Universal Robots PolyScope program: 2024DragonThinMarker.urp

Program 2024DragonThinMarker (installation=default directory=/programs createdIn=5.11.9.1010452 lastSavedIn=5.11.9.1010452 robotSerialNumber=20225200364)
Calibrated DH parameters: a=[0.00002, -0.569483, -0.54992, -0.00001, -0.000036, 0]; d=[0.180894, -146.691669, 192.918669, -46.053088, 0.119778, 0.115602]; alpha=[1.571425, -0.001534, 0.003359, 1.568739, -1.571477, 0]; deltaTheta=[0, 0.376258, -0.101074, -0.275185, -0.000002, 0]
Robot Program (runOnlyOnce=true)
  Script file /programs/usbdisk/new-robot/2024Dagonv3_1_thin_marker_large_2.script
    | def Machining1():
    |   # Default parameters:
    |   global speed_ms = 0.3
    |   global speed_rads = 0.75
    |   global accel_mss = 3
    |   global accel_radss = 1.2
    |   global blend_radius_m = 0.001
    | 
    |   # Add subprograms here
    |   # Start of main program
    |   # Program generated by RoboDK v5.6.5 for UR10e on 12/01/2024 13:40:53
    |   # Using nominal kinematics.
    |   blend_radius_m = 0.000
    |   speed_ms = 1.000
    |   # set_reference(p[0.335000, -0.152000, -0.010500, 0.000000, 0.000000, 0.000000])
    |   set_tcp(p[0.000000, 0.000000, 0.252000, 0.000000, 0.000000, 0.000000])
    |   # Show Tool
    |   movej([0.067194, -1.003010, -2.503941, -1.205438, 1.570796, 1.637990],accel_radss,speed_rads,0,blend_radius_m)
    |   movel([0.067194, -1.003010, -2.503941, -1.205438, 1.570796, 1.637990],accel_mss,speed_ms,0,blend_radius_m)
    |   # Splitting Linear movement in 22 (instruction 7: MoveL 3)
    |   movel([0.067194, -1.007550, -2.510737, -1.194102, 1.570796, 1.637990],accel_mss,speed_ms,0,blend_radius_m)
    |   movel([0.067194, -1.012266, -2.517496, -1.182627, 1.570796, 1.637990],accel_mss,speed_ms,0,blend_radius_m)
    |   movel([0.067194, -1.017163, -2.524216, -1.171010, 1.570796, 1.637990],accel_mss,speed_ms,0,blend_radius_m)
    |   movel([0.067194, -1.022245, -2.530898, -1.159246, 1.570796, 1.637990],accel_mss,speed_ms,0,blend_radius_m)
    |   movel([0.067194, -1.027517, -2.537540, -1.147332, 1.570796, 1.637990],accel_mss,speed_ms,0,blend_radius_m)
    |   movel([0.067194, -1.032983, -2.544142, -1.135264, 1.570796, 1.637990],accel_mss,speed_ms,0,blend_radius_m)
    |   movel([0.067194, -1.038648, -2.550703, -1.123038, 1.570796, 1.637990],accel_mss,speed_ms,0,blend_radius_m)
    |   movel([0.067194, -1.044517, -2.557222, -1.110650, 1.570796, 1.637990],accel_mss,speed_ms,0,blend_radius_m)
    |   movel([0.067194, -1.050595, -2.563697, -1.098097, 1.570796, 1.637990],accel_mss,speed_ms,0,blend_radius_m)
    |   movel([0.067194, -1.056888, -2.570128, -1.085374, 1.570796, 1.637990],accel_mss,speed_ms,0,blend_radius_m)
    |   movel([0.067194, -1.063399, -2.576514, -1.072476, 1.570796, 1.637990],accel_mss,speed_ms,0,blend_radius_m)
    |   movel([0.067194, -1.070135, -2.582853, -1.059401, 1.570796, 1.637990],accel_mss,speed_ms,0,blend_radius_m)
    |   movel([0.067194, -1.077101, -2.589145, -1.046144, 1.570796, 1.637990],accel_mss,speed_ms,0,blend_radius_m)
    |   movel([0.067194, -1.084302, -2.595388, -1.032699, 1.570796, 1.637990],accel_mss,speed_ms,0,blend_radius_m)
    |   movel([0.067194, -1.091744, -2.601581, -1.019064, 1.570796, 1.637990],accel_mss,speed_ms,0,blend_radius_m)
    |   movel([0.067194, -1.099433, -2.607722, -1.005234, 1.570796, 1.637990],accel_mss,speed_ms,0,blend_radius_m)
    |   movel([0.067194, -1.107374, -2.613811, -0.991204, 1.570796, 1.637990],accel_mss,speed_ms,0,blend_radius_m)
    |   movel([0.067194, -1.115573, -2.619846, -0.976970, 1.570796, 1.637990],accel_mss,speed_ms,0,blend_radius_m)
    |   movel([0.067194, -1.124036, -2.625825, -0.962528, 1.570796, 1.637990],accel_mss,speed_ms,0,blend_radius_m)
    |   movel([0.067194, -1.132769, -2.631747, -0.947873, 1.570796, 1.637990],accel_mss,speed_ms,0,blend_radius_m)
    |   movel([0.067194, -1.141778, -2.637610, -0.933001, 1.570796, 1.637990],accel_mss,speed_ms,0,blend_radius_m)
    |   movel([0.067194, -1.151068, -2.643412, -0.917908, 1.570796, 1.637990],accel_mss,speed_ms,0,blend_radius_m)
    |   movel([0.067194, -1.151068, -2.643412, -0.917908, 1.570796, 1.637990],accel_mss,speed_ms,0,blend_radius_m)
    |   speed_ms = 1.000
    |   movel([0.067194, -1.151068, -2.643412, -0.917908, 1.570796, 1.637990],accel_mss,speed_ms,0,blend_radius_m)
    |   movel([0.067194, -1.151068, -2.643412, -0.917908, 1.570796, 1.637990],accel_mss,speed_ms,0,blend_radius_m)
    |   movel([0.067194, -1.151068, -2.643412, -0.917908, 1.570796, 1.637990],accel_mss,speed_ms,0,blend_radius_m)
    |   speed_ms = 0.005
    |   # Splitting Linear movement in 4 (instruction 14: MoveL 8)
    |   movel([0.067194, -1.140864, -2.637026, -0.934498, 1.570796, 1.637990],accel_mss,speed_ms,0,blend_radius_m)
    |   movel([0.067194, -1.131001, -2.630567, -0.950821, 1.570796, 1.637990],accel_mss,speed_ms,0,blend_radius_m)
    |   movel([0.067194, -1.121469, -2.624037, -0.966883, 1.570796, 1.637990],accel_mss,speed_ms,0,blend_radius_m)
    |   movel([0.067194, -1.112262, -2.617439, -0.982688, 1.570796, 1.637990],accel_mss,speed_ms,0,blend_radius_m)
    |   speed_ms = 1.000
    |   # Splitting Linear movement in 4 (instruction 16: MoveL 9)
    |   movel([0.067194, -1.121469, -2.624037, -0.966883, 1.570796, 1.637990],accel_mss,speed_ms,0,blend_radius_m)
    |   movel([0.067194, -1.131001, -2.630567, -0.950821, 1.570796, 1.637990],accel_mss,speed_ms,0,blend_radius_m)
    |   movel([0.067194, -1.140864, -2.637026, -0.934498, 1.570796, 1.637990],accel_mss,speed_ms,0,blend_radius_m)
    |   movel([0.067194, -1.151068, -2.643412, -0.917908, 1.570796, 1.637990],accel_mss,speed_ms,0,blend_radius_m)
    |   speed_ms = 0.040
    |   movel([0.067194, -1.151068, -2.643412, -0.917908, 1.570796, 1.637990],accel_mss,speed_ms,0,blend_radius_m)
    |   speed_ms = 1.000
    |   movel([0.067194, -1.151068, -2.643412, -0.917908, 1.570796, 1.637990],accel_mss,speed_ms,0,blend_radius_m)
    |   # Splitting Linear movement in 16 (instruction 21: MoveL 12)
    |   movel([0.074500, -1.158538, -2.640023, -0.913828, 1.570796, 1.645297],accel_mss,speed_ms,0,blend_radius_m)
    |   movel([0.081655, -1.166054, -2.636556, -0.909779, 1.570796, 1.652452],accel_mss,speed_ms,0,blend_radius_m)
    |   movel([0.088662, -1.173611, -2.633012, -0.905766, 1.570796, 1.659459],accel_mss,speed_ms,0,blend_radius_m)
    |   movel([0.095525, -1.181205, -2.629391, -0.901793, 1.570796, 1.666321],accel_mss,speed_ms,0,blend_radius_m)
    |   movel([0.102245, -1.188830, -2.625693, -0.897865, 1.570796, 1.673041],accel_mss,speed_ms,0,blend_radius_m)
    |   movel([0.108826, -1.196483, -2.621921, -0.893985, 1.570796, 1.679622],accel_mss,speed_ms,0,blend_radius_m)
    |   movel([0.115271, -1.204158, -2.618073, -0.890157, 1.570796, 1.686068],accel_mss,speed_ms,0,blend_radius_m)
    |   movel([0.121584, -1.211853, -2.614152, -0.886384, 1.570796, 1.692381],accel_mss,speed_ms,0,blend_radius_m)
    |   movel([0.127767, -1.219562, -2.610158, -0.882669, 1.570796, 1.698563],accel_mss,speed_ms,0,blend_radius_m)
    |   movel([0.133823, -1.227283, -2.606091, -0.879015, 1.570796, 1.704619],accel_mss,speed_ms,0,blend_radius_m)
    |   movel([0.139755, -1.235012, -2.601952, -0.875425, 1.570796, 1.710551],accel_mss,speed_ms,0,blend_radius_m)
    |   movel([0.145566, -1.242745, -2.597743, -0.871901, 1.570796, 1.716362],accel_mss,speed_ms,0,blend_radius_m)
    |   movel([0.151258, -1.250480, -2.593464, -0.868445, 1.570796, 1.722054],accel_mss,speed_ms,0,blend_radius_m)
    |   movel([0.156835, -1.258213, -2.589116, -0.865060, 1.570796, 1.727631],accel_mss,speed_ms,0,blend_radius_m)
    |   movel([0.162299, -1.265943, -2.584700, -0.861746, 1.570796, 1.733095],accel_mss,speed_ms,0,blend_radius_m)
    |   movel([0.167652, -1.273666, -2.580216, -0.858507, 1.570796, 1.738448],accel_mss,speed_ms,0,blend_radius_m)
    |   speed_ms = 0.005
    |   # Splitting Linear movement in 4 (instruction 23: MoveL 13)
    |   movel([0.167652, -1.283824, -2.585872, -0.842693, 1.570796, 1.738448],accel_mss,speed_ms,0,blend_radius_m)
    |   movel([0.167652, -1.294258, -2.591445, -0.826686, 1.570796, 1.738448],accel_mss,speed_ms,0,blend_radius_m)
    |   movel([0.167652, -1.304973, -2.596930, -0.810486, 1.570796, 1.738448],accel_mss,speed_ms,0,blend_radius_m)
    |   movel([0.167652, -1.315971, -2.602326, -0.794092, 1.570796, 1.738448],accel_mss,speed_ms,0,blend_radius_m)
    |   speed_ms = 0.035
    |   movel([0.173157, -1.309286, -2.606449, -0.796654, 1.570796, 1.743953],accel_mss,speed_ms,0,blend_radius_m)
    |   movel([0.180818, -1.304394, -2.609429, -0.798566, 1.570796, 1.751614],accel_mss,speed_ms,0,blend_radius_m)
    |   movel([0.187193, -1.302810, -2.610387, -0.799192, 1.570796, 1.757989],accel_mss,speed_ms,0,blend_radius_m)
    |   movel([0.192434, -1.303607, -2.609905, -0.798877, 1.570796, 1.763230],accel_mss,speed_ms,0,blend_radius_m)
    |   movel([0.197299, -1.311355, -2.605179, -0.795855, 1.570796, 1.768095],accel_mss,speed_ms,0,blend_radius_m)
    |   movel([0.196080, -1.317152, -2.601592, -0.793645, 1.570796, 1.766876],accel_mss,speed_ms,0,blend_radius_m)
    |   movel([0.187692, -1.327691, -2.594957, -0.789741, 1.570796, 1.758489],accel_mss,speed_ms,0,blend_radius_m)
    |   movel([0.181558, -1.331218, -2.592703, -0.788467, 1.570796, 1.752354],accel_mss,speed_ms,0,blend_radius_m)
    |   movel([0.173175, -1.332644, -2.591788, -0.787957, 1.570796, 1.743971],accel_mss,speed_ms,0,blend_radius_m)
    |   speed_ms = 0.005
    |   movel([0.173175, -1.323918, -2.587552, -0.800919, 1.570796, 1.743971],accel_mss,speed_ms,0,blend_radius_m)
    |   speed_ms = 0.040
    |   # Splitting Linear movement in 4 (instruction 37: MoveL 24)
    |   movel([0.168800, -1.330792, -2.583155, -0.798442, 1.570796, 1.739596],accel_mss,speed_ms,0,blend_radius_m)
    |   movel([0.164486, -1.337594, -2.578742, -0.796052, 1.570796, 1.735282],accel_mss,speed_ms,0,blend_radius_m)
    |   movel([0.160232, -1.344326, -2.574314, -0.793749, 1.570796, 1.731029],accel_mss,speed_ms,0,blend_radius_m)
    |   movel([0.156038, -1.350989, -2.569871, -0.791529, 1.570796, 1.726834],accel_mss,speed_ms,0,blend_radius_m)
    |   speed_ms = 0.005
    |   movel([0.156038, -1.359551, -2.573989, -0.778848, 1.570796, 1.726834],accel_mss,speed_ms,0,blend_radius_m)
    |   speed_ms = 0.035
    |   movel([0.156883, -1.369330, -2.567274, -0.775785, 1.570796, 1.727679],accel_mss,speed_ms,0,blend_radius_m)
    |   movel([0.154042, -1.379446, -2.560185, -0.772758, 1.570796, 1.724839],accel_mss,speed_ms,0,blend_radius_m)
    |   movel([0.147953, -1.388965, -2.553382, -0.770042, 1.570796, 1.718749],accel_mss,speed_ms,0,blend_radius_m)
    |   movel([0.138991, -1.397044, -2.547506, -0.767839, 1.570796, 1.709787],accel_mss,speed_ms,0,blend_radius_m)
    |   movel([0.127521, -1.402604, -2.543408, -0.766378, 1.570796, 1.698317],accel_mss,speed_ms,0,blend_radius_m)
    |   movel([0.118961, -1.405060, -2.541583, -0.765746, 1.570796, 1.689757],accel_mss,speed_ms,0,blend_radius_m)
    |   speed_ms = 0.005
    |   movel([0.118961, -1.396797, -2.537660, -0.777932, 1.570796, 1.689757],accel_mss,speed_ms,0,blend_radius_m)
    |   speed_ms = 0.040
    |   # Splitting Linear movement in 2 (instruction 50: MoveL 33)
    |   movel([0.112287, -1.401146, -2.534448, -0.776795, 1.570796, 1.683083],accel_mss,speed_ms,0,blend_radius_m)
    |   movel([0.105663, -1.405490, -2.531212, -0.775687, 1.570796, 1.676460],accel_mss,speed_ms,0,blend_radius_m)
    |   speed_ms = 0.005
    |   movel([0.105663, -1.413694, -2.535098, -0.763597, 1.570796, 1.676460],accel_mss,speed_ms,0,blend_radius_m)
    |   speed_ms = 0.035
    |   movel([0.101650, -1.423004, -2.527983, -0.761402, 1.570796, 1.672447],accel_mss,speed_ms,0,blend_radius_m)
    |   movel([0.104946, -1.429410, -2.523012, -0.759967, 1.570796, 1.675742],accel_mss,speed_ms,0,blend_radius_m)
    |   movel([0.113388, -1.430242, -2.522362, -0.759785, 1.570796, 1.684184],accel_mss,speed_ms,0,blend_radius_m)
    |   movel([0.118946, -1.427701, -2.524344, -0.760344, 1.570796, 1.689742],accel_mss,speed_ms,0,blend_radius_m)
    |   movel([0.125116, -1.422682, -2.528231, -0.761476, 1.570796, 1.695912],accel_mss,speed_ms,0,blend_radius_m)
    |   speed_ms = 0.005
    |   movel([0.125116, -1.414541, -2.524382, -0.773466, 1.570796, 1.695912],accel_mss,speed_ms,0,blend_radius_m)
    |   speed_ms = 0.040
    |   # Splitting Linear movement in 6 (instruction 62: MoveL 41)
    |   movel([0.131385, -1.420188, -2.520061, -0.772140, 1.570796, 1.702182],accel_mss,speed_ms,0,blend_radius_m)
    |   movel([0.137555, -1.425859, -2.515674, -0.770856, 1.570796, 1.708351],accel_mss,speed_ms,0,blend_radius_m)
    |   movel([0.143625, -1.431553, -2.511222, -0.769614, 1.570796, 1.714422],accel_mss,speed_ms,0,blend_radius_m)
    |   movel([0.149599, -1.437267, -2.506705, -0.768417, 1.570796, 1.720395],accel_mss,speed_ms,0,blend_radius_m)
    |   movel([0.155477, -1.443000, -2.502125, -0.767263, 1.570796, 1.726274],accel_mss,speed_ms,0,blend_radius_m)
    |   movel([0.161262, -1.448750, -2.497482, -0.766156, 1.570796, 1.732058],accel_mss,speed_ms,0,blend_radius_m)
    |   speed_ms = 0.005
    |   movel([0.161262, -1.456649, -2.501190, -0.754550, 1.570796, 1.732058],accel_mss,speed_ms,0,blend_radius_m)
    |   speed_ms = 0.035
    |   # Splitting Linear movement in 4 (instruction 66: MoveL 43)
    |   movel([0.152429, -1.458352, -2.499789, -0.754248, 1.570796, 1.723226],accel_mss,speed_ms,0,blend_radius_m)
    |   movel([0.143603, -1.460114, -2.498334, -0.753941, 1.570796, 1.714400],accel_mss,speed_ms,0,blend_radius_m)
    |   movel([0.134785, -1.461934, -2.496827, -0.753628, 1.570796, 1.705581],accel_mss,speed_ms,0,blend_radius_m)
    |   movel([0.125976, -1.463810, -2.495267, -0.753312, 1.570796, 1.696772],accel_mss,speed_ms,0,blend_radius_m)
    |   # Splitting Linear movement in 4 (instruction 67: MoveL 44)
    |   movel([0.130374, -1.457124, -2.500800, -0.754465, 1.570796, 1.701171],accel_mss,speed_ms,0,blend_radius_m)
    |   movel([0.134837, -1.450374, -2.506316, -0.755698, 1.570796, 1.705633],accel_mss,speed_ms,0,blend_radius_m)
    |   movel([0.139366, -1.443560, -2.511816, -0.757013, 1.570796, 1.710162],accel_mss,speed_ms,0,blend_radius_m)
    |   movel([0.143961, -1.436680, -2.517298, -0.758412, 1.570796, 1.714758],accel_mss,speed_ms,0,blend_radius_m)
    |   movel([0.147089, -1.433429, -2.519863, -0.759097, 1.570796, 1.717886],accel_mss,speed_ms,0,blend_radius_m)
    |   movel([0.150947, -1.432131, -2.520882, -0.759376, 1.570796, 1.721743],accel_mss,speed_ms,0,blend_radius_m)
    |   movel([0.155136, -1.432926, -2.520258, -0.759205, 1.570796, 1.725933],accel_mss,speed_ms,0,blend_radius_m)
    |   movel([0.156013, -1.436691, -2.517289, -0.758410, 1.570796, 1.726809],accel_mss,speed_ms,0,blend_radius_m)
    |   # Splitting Linear movement in 2 (instruction 72: MoveL 49)
    |   movel([0.154617, -1.445524, -2.510238, -0.756627, 1.570796, 1.725413],accel_mss,speed_ms,0,blend_radius_m)
    |   movel([0.153250, -1.454249, -2.503159, -0.754982, 1.570796, 1.724046],accel_mss,speed_ms,0,blend_radius_m)
    |   speed_ms = 0.005
    |   movel([0.153250, -1.446333, -2.499441, -0.766616, 1.570796, 1.724046],accel_mss,speed_ms,0,blend_radius_m)
    |   speed_ms = 0.040
    |   # Splitting Linear movement in 4 (instruction 76: MoveL 51)
    |   movel([0.146625, -1.442667, -2.502393, -0.767329, 1.570796, 1.717422],accel_mss,speed_ms,0,blend_radius_m)
    |   movel([0.139925, -1.439047, -2.505289, -0.768053, 1.570796, 1.710722],accel_mss,speed_ms,0,blend_radius_m)
    |   movel([0.133149, -1.435473, -2.508129, -0.768787, 1.570796, 1.703945],accel_mss,speed_ms,0,blend_radius_m)
    |   movel([0.126295, -1.431947, -2.510912, -0.769530, 1.570796, 1.697092],accel_mss,speed_ms,0,blend_radius_m)
    |   speed_ms = 0.005
    |   movel([0.126295, -1.439966, -2.514688, -0.757735, 1.570796, 1.697092],accel_mss,speed_ms,0,blend_radius_m)
    |   speed_ms = 0.035
    |   # Splitting Linear movement in 4 (instruction 80: MoveL 53)
    |   movel([0.120303, -1.448950, -2.507472, -0.755967, 1.570796, 1.691099],accel_mss,speed_ms,0,blend_radius_m)
    |   movel([0.114424, -1.457822, -2.500226, -0.754341, 1.570796, 1.685220],accel_mss,speed_ms,0,blend_radius_m)
    |   movel([0.108656, -1.466585, -2.492951, -0.752853, 1.570796, 1.679453],accel_mss,speed_ms,0,blend_radius_m)
    |   movel([0.102997, -1.475244, -2.485647, -0.751498, 1.570796, 1.673793],accel_mss,speed_ms,0,blend_radius_m)
    |   speed_ms = 0.005
    |   movel([0.102997, -1.467481, -2.482014, -0.762894, 1.570796, 1.673793],accel_mss,speed_ms,0,blend_radius_m)
    |   speed_ms = 0.040
    |   movel([0.108909, -1.471851, -2.478329, -0.762209, 1.570796, 1.679706],accel_mss,speed_ms,0,blend_radius_m)
    |   speed_ms = 0.005
    |   movel([0.108909, -1.479582, -2.481945, -0.750863, 1.570796, 1.679706],accel_mss,speed_ms,0,blend_radius_m)
    |   speed_ms = 0.035
    |   # Splitting Linear movement in 6 (instruction 88: MoveL 57)
    |   movel([0.117333, -1.477702, -2.483553, -0.751135, 1.570796, 1.688130],accel_mss,speed_ms,0,blend_radius_m)
    |   movel([0.125768, -1.475873, -2.485112, -0.751404, 1.570796, 1.696564],accel_mss,speed_ms,0,blend_radius_m)
    |   movel([0.134212, -1.474095, -2.486622, -0.751671, 1.570796, 1.705008],accel_mss,speed_ms,0,blend_radius_m)
    |   movel([0.142664, -1.472370, -2.488083, -0.751935, 1.570796, 1.713461],accel_mss,speed_ms,0,blend_radius_m)
    |   movel([0.151124, -1.470699, -2.489495, -0.752195, 1.570796, 1.721920],accel_mss,speed_ms,0,blend_radius_m)
    |   movel([0.159589, -1.469080, -2.490858, -0.752451, 1.570796, 1.730386],accel_mss,speed_ms,0,blend_radius_m)
    |   speed_ms = 0.005
    |   movel([0.159589, -1.461273, -2.487200, -0.763916, 1.570796, 1.730386],accel_mss,speed_ms,0,blend_radius_m)
    |   speed_ms = 0.040
    |   movel([0.149536, -1.467349, -2.482125, -0.762915, 1.570796, 1.720332],accel_mss,speed_ms,0,blend_radius_m)
    |   speed_ms = 0.005
    |   movel([0.149536, -1.475113, -2.485758, -0.751518, 1.570796, 1.720332],accel_mss,speed_ms,0,blend_radius_m)
    |   speed_ms = 0.035
    |   # Splitting Linear movement in 2 (instruction 96: MoveL 61)
    |   movel([0.148238, -1.482664, -2.479296, -0.750429, 1.570796, 1.719034],accel_mss,speed_ms,0,blend_radius_m)
    |   movel([0.146962, -1.490139, -2.472812, -0.749438, 1.570796, 1.717758],accel_mss,speed_ms,0,blend_radius_m)
    |   speed_ms = 0.005
    |   movel([0.146962, -1.482487, -2.469238, -0.760664, 1.570796, 1.717758],accel_mss,speed_ms,0,blend_radius_m)
    |   speed_ms = 0.040
    |   # Splitting Linear movement in 4 (instruction 100: MoveL 63)
    |   movel([0.148044, -1.489667, -2.463003, -0.759718, 1.570796, 1.718840],accel_mss,speed_ms,0,blend_radius_m)
    |   movel([0.149106, -1.496792, -2.456739, -0.758858, 1.570796, 1.719903],accel_mss,speed_ms,0,blend_radius_m)
    |   movel([0.150151, -1.503862, -2.450444, -0.758082, 1.570796, 1.720947],accel_mss,speed_ms,0,blend_radius_m)
    |   movel([0.151177, -1.510880, -2.444121, -0.757388, 1.570796, 1.721973],accel_mss,speed_ms,0,blend_radius_m)
    |   speed_ms = 0.005
    |   movel([0.151177, -1.518320, -2.447586, -0.746483, 1.570796, 1.721973],accel_mss,speed_ms,0,blend_radius_m)
    |   speed_ms = 0.035
    |   movel([0.144185, -1.518298, -2.447607, -0.746484, 1.570796, 1.714981],accel_mss,speed_ms,0,blend_radius_m)
    |   movel([0.135810, -1.523039, -2.443241, -0.746109, 1.570796, 1.706606],accel_mss,speed_ms,0,blend_radius_m)
    |   speed_ms = 0.005
    |   movel([0.135810, -1.515634, -2.439793, -0.756962, 1.570796, 1.706606],accel_mss,speed_ms,0,blend_radius_m)
    |   speed_ms = 0.040
    |   # Splitting Linear movement in 2 (instruction 109: MoveL 68)
    |   movel([0.131950, -1.512601, -2.442559, -0.757230, 1.570796, 1.702747],accel_mss,speed_ms,0,blend_radius_m)
    |   movel([0.128057, -1.509579, -2.445299, -0.757511, 1.570796, 1.698854],accel_mss,speed_ms,0,blend_radius_m)
    |   speed_ms = 0.005
    |   movel([0.128057, -1.517029, -2.448769, -0.746591, 1.570796, 1.698854],accel_mss,speed_ms,0,blend_radius_m)
    |   speed_ms = 0.035
    |   movel([0.135688, -1.510985, -2.454272, -0.747132, 1.570796, 1.706484],accel_mss,speed_ms,0,blend_radius_m)
    |   movel([0.145709, -1.507599, -2.457330, -0.747461, 1.570796, 1.716505],accel_mss,speed_ms,0,blend_radius_m)
    |   movel([0.153057, -1.507247, -2.457646, -0.747496, 1.570796, 1.723854],accel_mss,speed_ms,0,blend_radius_m)
    |   movel([0.160779, -1.504715, -2.459919, -0.747754, 1.570796, 1.731575],accel_mss,speed_ms,0,blend_radius_m)
    |   movel([0.165697, -1.498711, -2.465270, -0.748408, 1.570796, 1.736494],accel_mss,speed_ms,0,blend_radius_m)
    |   movel([0.165769, -1.494615, -2.468888, -0.748886, 1.570796, 1.736565],accel_mss,speed_ms,0,blend_radius_m)
    |   movel([0.161795, -1.491118, -2.471957, -0.749314, 1.570796, 1.732592],accel_mss,speed_ms,0,blend_radius_m)
    |   speed_ms = 0.005
    |   movel([0.161795, -1.483474, -2.468386, -0.760529, 1.570796, 1.732592],accel_mss,speed_ms,0,blend_radius_m)
    |   speed_ms = 0.040
    |   movel([0.163598, -1.478856, -2.472361, -0.761172, 1.570796, 1.734394],accel_mss,speed_ms,0,blend_radius_m)
    |   speed_ms = 0.005
    |   movel([0.163598, -1.486535, -2.475950, -0.749905, 1.570796, 1.734394],accel_mss,speed_ms,0,blend_radius_m)
    |   speed_ms = 0.035
    |   # Splitting Linear movement in 6 (instruction 127: MoveL 80)
    |   movel([0.165237, -1.477873, -2.483407, -0.751110, 1.570796, 1.736033],accel_mss,speed_ms,0,blend_radius_m)
    |   movel([0.166909, -1.469106, -2.490836, -0.752447, 1.570796, 1.737705],accel_mss,speed_ms,0,blend_radius_m)
    |   movel([0.168617, -1.460232, -2.498236, -0.753920, 1.570796, 1.739413],accel_mss,speed_ms,0,blend_radius_m)
    |   movel([0.170360, -1.451246, -2.505608, -0.755535, 1.570796, 1.741157],accel_mss,speed_ms,0,blend_radius_m)
    |   movel([0.172141, -1.442144, -2.512950, -0.757295, 1.570796, 1.742938],accel_mss,speed_ms,0,blend_radius_m)
    |   movel([0.173961, -1.432921, -2.520262, -0.759206, 1.570796, 1.744757],accel_mss,speed_ms,0,blend_radius_m)
    |   movel([0.174121, -1.425301, -2.526207, -0.760881, 1.570796, 1.744918],accel_mss,speed_ms,0,blend_radius_m)
    |   movel([0.171855, -1.420034, -2.530266, -0.762089, 1.570796, 1.742651],accel_mss,speed_ms,0,blend_radius_m)
    |   movel([0.164710, -1.415086, -2.534042, -0.763261, 1.570796, 1.735506],accel_mss,speed_ms,0,blend_radius_m)
    |   movel([0.157581, -1.414562, -2.534440, -0.763387, 1.570796, 1.728377],accel_mss,speed_ms,0,blend_radius_m)
    |   movel([0.149868, -1.416547, -2.532931, -0.762911, 1.570796, 1.720665],accel_mss,speed_ms,0,blend_radius_m)
    |   # Splitting Linear movement in 2 (instruction 133: MoveL 86)
    |   movel([0.143461, -1.420629, -2.529810, -0.761950, 1.570796, 1.714257],accel_mss,speed_ms,0,blend_radius_m)
    |   movel([0.137100, -1.424708, -2.526667, -0.761015, 1.570796, 1.707896],accel_mss,speed_ms,0,blend_radius_m)
    |   # Splitting Linear movement in 2 (instruction 134: MoveL 87)
    |   movel([0.131353, -1.430632, -2.522057, -0.759700, 1.570796, 1.702149],accel_mss,speed_ms,0,blend_radius_m)
    |   movel([0.125674, -1.436514, -2.517428, -0.758446, 1.570796, 1.696470],accel_mss,speed_ms,0,blend_radius_m)
    |   movel([0.119296, -1.440811, -2.514015, -0.757564, 1.570796, 1.690092],accel_mss,speed_ms,0,blend_radius_m)
    |   movel([0.110431, -1.444256, -2.511257, -0.756876, 1.570796, 1.681228],accel_mss,speed_ms,0,blend_radius_m)
    |   movel([0.101817, -1.445410, -2.510330, -0.756649, 1.570796, 1.672613],accel_mss,speed_ms,0,blend_radius_m)
    |   movel([0.094928, -1.444091, -2.511390, -0.756908, 1.570796, 1.665724],accel_mss,speed_ms,0,blend_radius_m)
    |   # Splitting Linear movement in 2 (instruction 139: MoveL 92)
    |   movel([0.090922, -1.441165, -2.513732, -0.757492, 1.570796, 1.661719],accel_mss,speed_ms,0,blend_radius_m)
    |   movel([0.086882, -1.438253, -2.516050, -0.758086, 1.570796, 1.657679],accel_mss,speed_ms,0,blend_radius_m)
    |   # Splitting Linear movement in 2 (instruction 140: MoveL 93)
    |   movel([0.085417, -1.432512, -2.520583, -0.759294, 1.570796, 1.656214],accel_mss,speed_ms,0,blend_radius_m)
    |   movel([0.083931, -1.426737, -2.525094, -0.760558, 1.570796, 1.654728],accel_mss,speed_ms,0,blend_radius_m)
    |   # Splitting Linear movement in 2 (instruction 141: MoveL 94)
    |   movel([0.085999, -1.420689, -2.529764, -0.761936, 1.570796, 1.656796],accel_mss,speed_ms,0,blend_radius_m)
    |   movel([0.088096, -1.414585, -2.534422, -0.763381, 1.570796, 1.658892],accel_mss,speed_ms,0,blend_radius_m)
    |   # Splitting Linear movement in 2 (instruction 142: MoveL 95)
    |   movel([0.092936, -1.409123, -2.538545, -0.764721, 1.570796, 1.663732],accel_mss,speed_ms,0,blend_radius_m)
    |   movel([0.097830, -1.403621, -2.542653, -0.766115, 1.570796, 1.668626],accel_mss,speed_ms,0,blend_radius_m)
    |   # Splitting Linear movement in 2 (instruction 143: MoveL 96)
    |   movel([0.104573, -1.399755, -2.545513, -0.767121, 1.570796, 1.675370],accel_mss,speed_ms,0,blend_radius_m)
    |   movel([0.111360, -1.395891, -2.548350, -0.768147, 1.570796, 1.682157],accel_mss,speed_ms,0,blend_radius_m)
    |   speed_ms = 0.005
    |   movel([0.111360, -1.387566, -2.544389, -0.780434, 1.570796, 1.682157],accel_mss,speed_ms,0,blend_radius_m)
    |   speed_ms = 0.040
    |   movel([0.119864, -1.383368, -2.547408, -0.781612, 1.570796, 1.690661],accel_mss,speed_ms,0,blend_radius_m)
    |   speed_ms = 0.005
    |   movel([0.119864, -1.391722, -2.551388, -0.769280, 1.570796, 1.690661],accel_mss,speed_ms,0,blend_radius_m)
    |   speed_ms = 0.035
    |   movel([0.127885, -1.389591, -2.552930, -0.769868, 1.570796, 1.698681],accel_mss,speed_ms,0,blend_radius_m)
    |   movel([0.133367, -1.385898, -2.555588, -0.770903, 1.570796, 1.704163],accel_mss,speed_ms,0,blend_radius_m)
    |   movel([0.139947, -1.375961, -2.562643, -0.773785, 1.570796, 1.710744],accel_mss,speed_ms,0,blend_radius_m)
    |   movel([0.140218, -1.370886, -2.566192, -0.775310, 1.570796, 1.711014],accel_mss,speed_ms,0,blend_radius_m)
    |   movel([0.134172, -1.364852, -2.570365, -0.777171, 1.570796, 1.704969],accel_mss,speed_ms,0,blend_radius_m)
    |   movel([0.128886, -1.364770, -2.570422, -0.777197, 1.570796, 1.699682],accel_mss,speed_ms,0,blend_radius_m)
    |   movel([0.122870, -1.366828, -2.569005, -0.776556, 1.570796, 1.693666],accel_mss,speed_ms,0,blend_radius_m)
    |   movel([0.116129, -1.371828, -2.565537, -0.775024, 1.570796, 1.686926],accel_mss,speed_ms,0,blend_radius_m)
    |   movel([0.111791, -1.378110, -2.561130, -0.773150, 1.570796, 1.682587],accel_mss,speed_ms,0,blend_radius_m)
    |   speed_ms = 0.005
    |   movel([0.111791, -1.369666, -2.557092, -0.785631, 1.570796, 1.682587],accel_mss,speed_ms,0,blend_radius_m)
    |   speed_ms = 0.040
    |   # Splitting Linear movement in 2 (instruction 163: MoveL 110)
    |   movel([0.102143, -1.369221, -2.557402, -0.785766, 1.570796, 1.672940],accel_mss,speed_ms,0,blend_radius_m)
    |   movel([0.092446, -1.368873, -2.557645, -0.785872, 1.570796, 1.663242],accel_mss,speed_ms,0,blend_radius_m)
    |   speed_ms = 0.005
    |   movel([0.092446, -1.377321, -2.561686, -0.773382, 1.570796, 1.663242],accel_mss,speed_ms,0,blend_radius_m)
    |   speed_ms = 0.035
    |   # Splitting Linear movement in 2 (instruction 167: MoveL 112)
    |   movel([0.096801, -1.371069, -2.566066, -0.775255, 1.570796, 1.667598],accel_mss,speed_ms,0,blend_radius_m)
    |   movel([0.101214, -1.364757, -2.570431, -0.777201, 1.570796, 1.672011],accel_mss,speed_ms,0,blend_radius_m)
    |   movel([0.109892, -1.356186, -2.576270, -0.779933, 1.570796, 1.680688],accel_mss,speed_ms,0,blend_radius_m)
    |   # Splitting Linear movement in 2 (instruction 169: MoveL 114)
    |   movel([0.116564, -1.352214, -2.578941, -0.781234, 1.570796, 1.687360],accel_mss,speed_ms,0,blend_radius_m)
    |   movel([0.123279, -1.348242, -2.581591, -0.782556, 1.570796, 1.694075],accel_mss,speed_ms,0,blend_radius_m)
    |   # Splitting Linear movement in 2 (instruction 170: MoveL 115)
    |   movel([0.130460, -1.346443, -2.582783, -0.783162, 1.570796, 1.701256],accel_mss,speed_ms,0,blend_radius_m)
    |   movel([0.137648, -1.344681, -2.583948, -0.783760, 1.570796, 1.708444],accel_mss,speed_ms,0,blend_radius_m)
    |   # Splitting Linear movement in 2 (instruction 171: MoveL 116)
    |   movel([0.147112, -1.346959, -2.582442, -0.782988, 1.570796, 1.717908],accel_mss,speed_ms,0,blend_radius_m)
    |   movel([0.156484, -1.349338, -2.580862, -0.782189, 1.570796, 1.727280],accel_mss,speed_ms,0,blend_radius_m)
    |   movel([0.165265, -1.351727, -2.579267, -0.781395, 1.570796, 1.736061],accel_mss,speed_ms,0,blend_radius_m)
    |   movel([0.175465, -1.350957, -2.579782, -0.781650, 1.570796, 1.746261],accel_mss,speed_ms,0,blend_radius_m)
    |   movel([0.186285, -1.347233, -2.582261, -0.782896, 1.570796, 1.757082],accel_mss,speed_ms,0,blend_radius_m)
    |   movel([0.196943, -1.340710, -2.586556, -0.785123, 1.570796, 1.767739],accel_mss,speed_ms,0,blend_radius_m)
    |   movel([0.205914, -1.332349, -2.591977, -0.788062, 1.570796, 1.776710],accel_mss,speed_ms,0,blend_radius_m)
    |   movel([0.213309, -1.322133, -2.598475, -0.791782, 1.570796, 1.784105],accel_mss,speed_ms,0,blend_radius_m)
    |   movel([0.218019, -1.310769, -2.605539, -0.796081, 1.570796, 1.788815],accel_mss,speed_ms,0,blend_radius_m)
    |   movel([0.218847, -1.299039, -2.612655, -0.800695, 1.570796, 1.789643],accel_mss,speed_ms,0,blend_radius_m)
    |   movel([0.215629, -1.290767, -2.617567, -0.804055, 1.570796, 1.786426],accel_mss,speed_ms,0,blend_radius_m)
    |   movel([0.208938, -1.285368, -2.620726, -0.806295, 1.570796, 1.779735],accel_mss,speed_ms,0,blend_radius_m)
    |   movel([0.199486, -1.283243, -2.621959, -0.807187, 1.570796, 1.770282],accel_mss,speed_ms,0,blend_radius_m)
    |   movel([0.188071, -1.284713, -2.621106, -0.806569, 1.570796, 1.758867],accel_mss,speed_ms,0,blend_radius_m)
    |   movel([0.175553, -1.290033, -2.617999, -0.804358, 1.570796, 1.746349],accel_mss,speed_ms,0,blend_radius_m)
    |   movel([0.164105, -1.298333, -2.613078, -0.800978, 1.570796, 1.734901],accel_mss,speed_ms,0,blend_radius_m)
    |   movel([0.154717, -1.308660, -2.606832, -0.796897, 1.570796, 1.725514],accel_mss,speed_ms,0,blend_radius_m)
    |   movel([0.148273, -1.320113, -2.599743, -0.792533, 1.570796, 1.719069],accel_mss,speed_ms,0,blend_radius_m)
    |   speed_ms = 0.005
    |   movel([0.148273, -1.311314, -2.595451, -0.805623, 1.570796, 1.719069],accel_mss,speed_ms,0,blend_radius_m)
    |   speed_ms = 0.040
    |   movel([0.148587, -1.300615, -2.601996, -0.809778, 1.570796, 1.719384],accel_mss,speed_ms,0,blend_radius_m)
    |   speed_ms = 0.005
    |   movel([0.148587, -1.309472, -2.606335, -0.796582, 1.570796, 1.719384],accel_mss,speed_ms,0,blend_radius_m)
    |   speed_ms = 0.035
    |   # Splitting Linear movement in 2 (instruction 195: MoveL 136)
    |   movel([0.141454, -1.310148, -2.605920, -0.796320, 1.570796, 1.712250],accel_mss,speed_ms,0,blend_radius_m)
    |   movel([0.134308, -1.310872, -2.605476, -0.796041, 1.570796, 1.705104],accel_mss,speed_ms,0,blend_radius_m)
    |   # Splitting Linear movement in 2 (instruction 196: MoveL 137)
    |   movel([0.128832, -1.308947, -2.606656, -0.796786, 1.570796, 1.699629],accel_mss,speed_ms,0,blend_radius_m)
    |   movel([0.123318, -1.307057, -2.607810, -0.797521, 1.570796, 1.694114],accel_mss,speed_ms,0,blend_radius_m)
    |   # Splitting Linear movement in 2 (instruction 197: MoveL 138)
    |   movel([0.119974, -1.302841, -2.610368, -0.799180, 1.570796, 1.690770],accel_mss,speed_ms,0,blend_radius_m)
    |   movel([0.116592, -1.298625, -2.612903, -0.800861, 1.570796, 1.687388],accel_mss,speed_ms,0,blend_radius_m)
    |   # Splitting Linear movement in 2 (instruction 198: MoveL 139)
    |   movel([0.115954, -1.292359, -2.616628, -0.803402, 1.570796, 1.686750],accel_mss,speed_ms,0,blend_radius_m)
    |   movel([0.115306, -1.286042, -2.620333, -0.806014, 1.570796, 1.686102],accel_mss,speed_ms,0,blend_radius_m)
    |   # Splitting Linear movement in 2 (instruction 199: MoveL 140)
    |   movel([0.117736, -1.278694, -2.624580, -0.809115, 1.570796, 1.688532],accel_mss,speed_ms,0,blend_radius_m)
    |   movel([0.120205, -1.271258, -2.628809, -0.812322, 1.570796, 1.691002],accel_mss,speed_ms,0,blend_radius_m)
    |   # Splitting Linear movement in 2 (instruction 200: MoveL 141)
    |   movel([0.125251, -1.264165, -2.632779, -0.815444, 1.570796, 1.696048],accel_mss,speed_ms,0,blend_radius_m)
    |   movel([0.130370, -1.256992, -2.636733, -0.818665, 1.570796, 1.701166],accel_mss,speed_ms,0,blend_radius_m)
    |   # Splitting Linear movement in 2 (instruction 201: MoveL 142)
    |   movel([0.137370, -1.251001, -2.639986, -0.821401, 1.570796, 1.708167],accel_mss,speed_ms,0,blend_radius_m)
    |   movel([0.144445, -1.244971, -2.643219, -0.824200, 1.570796, 1.715241],accel_mss,speed_ms,0,blend_radius_m)
    |   # Splitting Linear movement in 2 (instruction 202: MoveL 143)
    |   movel([0.152629, -1.241031, -2.645307, -0.826051, 1.570796, 1.723426],accel_mss,speed_ms,0,blend_radius_m)
    |   movel([0.160854, -1.237110, -2.647367, -0.827911, 1.570796, 1.731651],accel_mss,speed_ms,0,blend_radius_m)
    |   # Splitting Linear movement in 2 (instruction 203: MoveL 144)
    |   movel([0.170134, -1.236501, -2.647686, -0.828202, 1.570796, 1.740930],accel_mss,speed_ms,0,blend_radius_m)
    |   movel([0.179381, -1.235980, -2.647958, -0.828451, 1.570796, 1.750178],accel_mss,speed_ms,0,blend_radius_m)
    |   speed_ms = 0.005
    |   movel([0.179381, -1.226775, -2.643291, -0.842324, 1.570796, 1.750178],accel_mss,speed_ms,0,blend_radius_m)
    |   speed_ms = 0.040
    |   # Splitting Linear movement in 4 (instruction 207: MoveL 146)
    |   movel([0.176492, -1.237455, -2.637721, -0.837213, 1.570796, 1.747289],accel_mss,speed_ms,0,blend_radius_m)
    |   movel([0.173670, -1.247958, -2.632114, -0.832317, 1.570796, 1.744466],accel_mss,speed_ms,0,blend_radius_m)
    |   movel([0.170910, -1.258290, -2.626471, -0.827627, 1.570796, 1.741707],accel_mss,speed_ms,0,blend_radius_m)
    |   movel([0.168213, -1.268457, -2.620794, -0.823138, 1.570796, 1.739009],accel_mss,speed_ms,0,blend_radius_m)
    |   speed_ms = 0.005
    |   movel([0.168213, -1.277479, -2.625275, -0.809634, 1.570796, 1.739009],accel_mss,speed_ms,0,blend_radius_m)
    |   speed_ms = 0.035
    |   movel([0.161916, -1.284229, -2.621387, -0.806772, 1.570796, 1.732712],accel_mss,speed_ms,0,blend_radius_m)
    |   movel([0.153892, -1.288752, -2.618750, -0.804887, 1.570796, 1.724689],accel_mss,speed_ms,0,blend_radius_m)
    |   movel([0.147527, -1.289906, -2.618073, -0.804410, 1.570796, 1.718324],accel_mss,speed_ms,0,blend_radius_m)
    |   movel([0.142466, -1.288702, -2.618780, -0.804908, 1.570796, 1.713263],accel_mss,speed_ms,0,blend_radius_m)
    |   movel([0.138212, -1.280197, -2.623717, -0.808475, 1.570796, 1.709008],accel_mss,speed_ms,0,blend_radius_m)
    |   movel([0.139872, -1.273980, -2.627269, -0.811140, 1.570796, 1.710668],accel_mss,speed_ms,0,blend_radius_m)
    |   movel([0.149427, -1.262659, -2.633614, -0.816115, 1.570796, 1.720224],accel_mss,speed_ms,0,blend_radius_m)
    |   movel([0.156179, -1.258999, -2.635633, -0.817757, 1.570796, 1.726975],accel_mss,speed_ms,0,blend_radius_m)
    |   movel([0.165037, -1.257988, -2.636188, -0.818214, 1.570796, 1.735834],accel_mss,speed_ms,0,blend_radius_m)
    |   speed_ms = 0.005
    |   movel([0.165037, -1.248875, -2.631619, -0.831896, 1.570796, 1.735834],accel_mss,speed_ms,0,blend_radius_m)
    |   speed_ms = 0.040
    |   movel([0.166836, -1.237491, -2.637702, -0.837196, 1.570796, 1.737632],accel_mss,speed_ms,0,blend_radius_m)
    |   speed_ms = 0.005
    |   movel([0.166836, -1.246653, -2.642321, -0.823414, 1.570796, 1.737632],accel_mss,speed_ms,0,blend_radius_m)
    |   speed_ms = 0.035
    |   # Splitting Linear movement in 2 (instruction 227: MoveL 160)
    |   movel([0.175033, -1.246326, -2.642496, -0.823567, 1.570796, 1.745829],accel_mss,speed_ms,0,blend_radius_m)
    |   movel([0.183201, -1.246069, -2.642633, -0.823687, 1.570796, 1.753998],accel_mss,speed_ms,0,blend_radius_m)
    |   movel([0.197166, -1.239847, -2.645931, -0.826611, 1.570796, 1.767962],accel_mss,speed_ms,0,blend_radius_m)
    |   movel([0.209753, -1.229814, -2.651154, -0.831421, 1.570796, 1.780549],accel_mss,speed_ms,0,blend_radius_m)
    |   movel([0.219721, -1.217088, -2.657611, -0.837690, 1.570796, 1.790517],accel_mss,speed_ms,0,blend_radius_m)
    |   movel([0.225661, -1.202884, -2.664603, -0.844902, 1.570796, 1.796457],accel_mss,speed_ms,0,blend_radius_m)
    |   movel([0.226421, -1.192028, -2.669797, -0.850564, 1.570796, 1.797217],accel_mss,speed_ms,0,blend_radius_m)
    |   movel([0.223372, -1.183529, -2.673774, -0.855086, 1.570796, 1.794168],accel_mss,speed_ms,0,blend_radius_m)
    |   movel([0.216908, -1.178001, -2.676320, -0.858068, 1.570796, 1.787704],accel_mss,speed_ms,0,blend_radius_m)
    |   movel([0.207511, -1.176027, -2.677221, -0.859141, 1.570796, 1.778307],accel_mss,speed_ms,0,blend_radius_m)
    |   speed_ms = 0.005
    |   movel([0.207511, -1.166631, -2.672286, -0.873473, 1.570796, 1.778307],accel_mss,speed_ms,0,blend_radius_m)
    |   speed_ms = 0.040
    |   # Splitting Linear movement in 2 (instruction 239: MoveL 170)
    |   movel([0.204969, -1.176006, -2.668022, -0.868361, 1.570796, 1.775765],accel_mss,speed_ms,0,blend_radius_m)
    |   movel([0.202477, -1.185246, -2.663729, -0.863414, 1.570796, 1.773273],accel_mss,speed_ms,0,blend_radius_m)
    |   speed_ms = 0.005
    |   movel([0.202477, -1.194593, -2.668581, -0.849214, 1.570796, 1.773273],accel_mss,speed_ms,0,blend_radius_m)
    |   speed_ms = 0.035
    |   movel([0.210010, -1.200039, -2.665977, -0.846373, 1.570796, 1.780806],accel_mss,speed_ms,0,blend_radius_m)
    |   movel([0.209614, -1.209388, -2.661430, -0.841571, 1.570796, 1.780410],accel_mss,speed_ms,0,blend_radius_m)
    |   movel([0.204605, -1.219143, -2.656581, -0.836665, 1.570796, 1.775402],accel_mss,speed_ms,0,blend_radius_m)
    |   movel([0.198126, -1.226077, -2.653069, -0.833243, 1.570796, 1.768923],accel_mss,speed_ms,0,blend_radius_m)
    |   speed_ms = 0.005
    |   movel([0.198126, -1.216834, -2.648358, -0.847198, 1.570796, 1.768923],accel_mss,speed_ms,0,blend_radius_m)
    |   speed_ms = 0.040
    |   # Splitting Linear movement in 4 (instruction 250: MoveL 177)
    |   movel([0.206150, -1.214385, -2.649588, -0.848415, 1.570796, 1.776946],accel_mss,speed_ms,0,blend_radius_m)
    |   movel([0.214184, -1.211979, -2.650791, -0.849618, 1.570796, 1.784980],accel_mss,speed_ms,0,blend_radius_m)
    |   movel([0.222229, -1.209617, -2.651966, -0.850806, 1.570796, 1.793025],accel_mss,speed_ms,0,blend_radius_m)
    |   movel([0.230283, -1.207299, -2.653113, -0.851977, 1.570796, 1.801080],accel_mss,speed_ms,0,blend_radius_m)
    |   speed_ms = 0.005
    |   movel([0.230283, -1.216576, -2.657867, -0.837946, 1.570796, 1.801080],accel_mss,speed_ms,0,blend_radius_m)
    |   speed_ms = 0.035
    |   movel([0.236227, -1.211381, -2.660448, -0.840560, 1.570796, 1.807024],accel_mss,speed_ms,0,blend_radius_m)
    |   movel([0.238365, -1.205658, -2.663256, -0.843476, 1.570796, 1.809161],accel_mss,speed_ms,0,blend_radius_m)
    |   movel([0.236377, -1.201779, -2.665138, -0.845472, 1.570796, 1.807173],accel_mss,speed_ms,0,blend_radius_m)
    |   movel([0.229957, -1.202188, -2.664940, -0.845261, 1.570796, 1.800753],accel_mss,speed_ms,0,blend_radius_m)
    |   speed_ms = 0.005
    |   movel([0.229957, -1.192864, -2.660122, -0.859404, 1.570796, 1.800753],accel_mss,speed_ms,0,blend_radius_m)
    |   speed_ms = 0.040
    |   # Splitting Linear movement in 2 (instruction 261: MoveL 184)
    |   movel([0.238588, -1.188973, -2.661972, -0.861444, 1.570796, 1.809384],accel_mss,speed_ms,0,blend_radius_m)
    |   movel([0.247256, -1.185109, -2.663793, -0.863487, 1.570796, 1.818052],accel_mss,speed_ms,0,blend_radius_m)
    |   speed_ms = 0.005
    |   movel([0.247256, -1.194457, -2.668646, -0.849286, 1.570796, 1.818052],accel_mss,speed_ms,0,blend_radius_m)
    |   speed_ms = 0.035
    |   movel([0.247940, -1.188279, -2.671561, -0.852549, 1.570796, 1.818737],accel_mss,speed_ms,0,blend_radius_m)
    |   movel([0.243895, -1.185291, -2.672956, -0.854142, 1.570796, 1.814691],accel_mss,speed_ms,0,blend_radius_m)
    |   movel([0.235099, -1.186707, -2.672296, -0.853386, 1.570796, 1.805895],accel_mss,speed_ms,0,blend_radius_m)
    |   movel([0.230944, -1.183872, -2.673615, -0.854902, 1.570796, 1.801741],accel_mss,speed_ms,0,blend_radius_m)
    |   movel([0.232076, -1.178742, -2.675980, -0.857667, 1.570796, 1.802873],accel_mss,speed_ms,0,blend_radius_m)
    |   movel([0.236326, -1.174585, -2.677876, -0.859927, 1.570796, 1.807122],accel_mss,speed_ms,0,blend_radius_m)
    |   movel([0.241419, -1.174801, -2.677779, -0.859810, 1.570796, 1.812215],accel_mss,speed_ms,0,blend_radius_m)
    |   speed_ms = 0.005
    |   movel([0.241419, -1.165402, -2.672838, -0.874149, 1.570796, 1.812215],accel_mss,speed_ms,0,blend_radius_m)
    |   speed_ms = 0.040
    |   # Splitting Linear movement in 4 (instruction 275: MoveL 194)
    |   movel([0.240761, -1.158708, -2.675818, -0.877863, 1.570796, 1.811558],accel_mss,speed_ms,0,blend_radius_m)
    |   movel([0.240093, -1.151960, -2.678777, -0.881653, 1.570796, 1.810890],accel_mss,speed_ms,0,blend_radius_m)
    |   movel([0.239415, -1.145155, -2.681713, -0.885520, 1.570796, 1.810211],accel_mss,speed_ms,0,blend_radius_m)
    |   movel([0.238725, -1.138295, -2.684628, -0.889467, 1.570796, 1.809521],accel_mss,speed_ms,0,blend_radius_m)
    |   speed_ms = 0.005
    |   movel([0.238725, -1.147747, -2.689688, -0.874954, 1.570796, 1.809521],accel_mss,speed_ms,0,blend_radius_m)
    |   speed_ms = 0.035
    |   # Splitting Linear movement in 2 (instruction 279: MoveL 196)
    |   movel([0.225987, -1.157432, -2.685510, -0.869447, 1.570796, 1.796784],accel_mss,speed_ms,0,blend_radius_m)
    |   movel([0.213438, -1.167038, -2.681273, -0.864078, 1.570796, 1.784234],accel_mss,speed_ms,0,blend_radius_m)
    |   # Splitting Linear movement in 4 (instruction 280: MoveL 197)
    |   movel([0.201011, -1.173908, -2.678183, -0.860297, 1.570796, 1.771808],accel_mss,speed_ms,0,blend_radius_m)
    |   movel([0.188695, -1.180794, -2.675038, -0.856557, 1.570796, 1.759491],accel_mss,speed_ms,0,blend_radius_m)
    |   movel([0.176490, -1.187692, -2.671836, -0.852861, 1.570796, 1.747286],accel_mss,speed_ms,0,blend_radius_m)
    |   movel([0.164397, -1.194600, -2.668578, -0.849211, 1.570796, 1.735193],accel_mss,speed_ms,0,blend_radius_m)
    |   speed_ms = 0.005
    |   movel([0.164397, -1.185253, -2.663726, -0.863410, 1.570796, 1.735193],accel_mss,speed_ms,0,blend_radius_m)
    |   speed_ms = 0.040
    |   movel([0.159806, -1.191461, -2.660791, -0.860138, 1.570796, 1.730603],accel_mss,speed_ms,0,blend_radius_m)
    |   speed_ms = 0.005
    |   movel([0.159806, -1.200789, -2.665616, -0.845984, 1.570796, 1.730603],accel_mss,speed_ms,0,blend_radius_m)
    |   speed_ms = 0.035
    |   movel([0.160903, -1.196857, -2.667503, -0.848030, 1.570796, 1.731700],accel_mss,speed_ms,0,blend_radius_m)
    |   movel([0.154429, -1.194191, -2.668773, -0.849426, 1.570796, 1.725225],accel_mss,speed_ms,0,blend_radius_m)
    |   movel([0.144721, -1.201195, -2.665420, -0.845774, 1.570796, 1.715517],accel_mss,speed_ms,0,blend_radius_m)
    |   movel([0.137954, -1.200037, -2.665978, -0.846374, 1.570796, 1.708750],accel_mss,speed_ms,0,blend_radius_m)
    |   movel([0.132182, -1.205574, -2.663297, -0.843519, 1.570796, 1.702978],accel_mss,speed_ms,0,blend_radius_m)
    |   movel([0.131588, -1.210593, -2.660837, -0.840959, 1.570796, 1.702385],accel_mss,speed_ms,0,blend_radius_m)
    |   speed_ms = 0.005
    |   movel([0.131588, -1.201296, -2.656055, -0.855038, 1.570796, 1.702385],accel_mss,speed_ms,0,blend_radius_m)
    |   speed_ms = 0.040
    |   # Splitting Linear movement in 2 (instruction 297: MoveL 208)
    |   movel([0.120746, -1.207729, -2.652901, -0.851759, 1.570796, 1.691542],accel_mss,speed_ms,0,blend_radius_m)
    |   movel([0.110002, -1.214162, -2.649700, -0.848527, 1.570796, 1.680798],accel_mss,speed_ms,0,blend_radius_m)
    |   speed_ms = 0.005
    |   movel([0.110002, -1.223415, -2.654424, -0.834550, 1.570796, 1.680798],accel_mss,speed_ms,0,blend_radius_m)
    |   speed_ms = 0.035
    |   movel([0.115547, -1.217819, -2.657245, -0.837324, 1.570796, 1.686344],accel_mss,speed_ms,0,blend_radius_m)
    |   movel([0.119180, -1.216467, -2.657922, -0.838000, 1.570796, 1.689976],accel_mss,speed_ms,0,blend_radius_m)
    |   movel([0.121294, -1.219629, -2.656337, -0.836423, 1.570796, 1.692091],accel_mss,speed_ms,0,blend_radius_m)
    |   movel([0.120048, -1.223191, -2.654538, -0.834660, 1.570796, 1.690844],accel_mss,speed_ms,0,blend_radius_m)
    |   movel([0.119326, -1.229089, -2.651527, -0.831774, 1.570796, 1.690122],accel_mss,speed_ms,0,blend_radius_m)
    |   movel([0.122415, -1.229575, -2.651277, -0.831537, 1.570796, 1.693211],accel_mss,speed_ms,0,blend_radius_m)
    |   movel([0.131972, -1.220221, -2.656039, -0.836129, 1.570796, 1.702768],accel_mss,speed_ms,0,blend_radius_m)
    |   movel([0.139556, -1.214277, -2.659013, -0.839099, 1.570796, 1.710353],accel_mss,speed_ms,0,blend_radius_m)
    |   movel([0.145156, -1.213265, -2.659515, -0.839609, 1.570796, 1.715952],accel_mss,speed_ms,0,blend_radius_m)
    |   speed_ms = 0.005
    |   movel([0.145156, -1.203977, -2.654746, -0.853666, 1.570796, 1.715952],accel_mss,speed_ms,0,blend_radius_m)
    |   speed_ms = 0.040
    |   movel([0.137408, -1.218124, -2.647706, -0.846559, 1.570796, 1.708204],accel_mss,speed_ms,0,blend_radius_m)
    |   speed_ms = 0.005
    |   movel([0.137408, -1.227362, -2.652412, -0.832615, 1.570796, 1.708204],accel_mss,speed_ms,0,blend_radius_m)
    |   speed_ms = 0.035
    |   movel([0.141534, -1.229933, -2.651092, -0.831364, 1.570796, 1.712331],accel_mss,speed_ms,0,blend_radius_m)
    |   movel([0.145013, -1.229003, -2.651571, -0.831815, 1.570796, 1.715809],accel_mss,speed_ms,0,blend_radius_m)
    |   movel([0.154603, -1.217032, -2.657639, -0.837718, 1.570796, 1.725399],accel_mss,speed_ms,0,blend_radius_m)
    |   movel([0.165974, -1.208279, -2.661974, -0.842136, 1.570796, 1.736771],accel_mss,speed_ms,0,blend_radius_m)
    |   movel([0.179620, -1.207005, -2.662598, -0.842786, 1.570796, 1.750416],accel_mss,speed_ms,0,blend_radius_m)
    |   movel([0.183761, -1.206444, -2.662872, -0.843073, 1.570796, 1.754557],accel_mss,speed_ms,0,blend_radius_m)
    |   movel([0.189391, -1.203031, -2.664532, -0.844826, 1.570796, 1.760187],accel_mss,speed_ms,0,blend_radius_m)
    |   movel([0.194299, -1.196782, -2.667538, -0.848068, 1.570796, 1.765095],accel_mss,speed_ms,0,blend_radius_m)
    |   movel([0.196243, -1.187663, -2.671849, -0.852876, 1.570796, 1.767039],accel_mss,speed_ms,0,blend_radius_m)
    |   speed_ms = 0.005
    |   movel([0.196243, -1.178297, -2.666966, -0.867126, 1.570796, 1.767039],accel_mss,speed_ms,0,blend_radius_m)
    |   speed_ms = 0.040
    |   movel([0.187393, -1.179350, -2.666479, -0.866560, 1.570796, 1.758189],accel_mss,speed_ms,0,blend_radius_m)
    |   speed_ms = 0.005
    |   movel([0.187393, -1.188714, -2.671357, -0.852318, 1.570796, 1.758189],accel_mss,speed_ms,0,blend_radius_m)
    |   speed_ms = 0.035
    |   movel([0.183829, -1.194575, -2.668590, -0.849224, 1.570796, 1.754625],accel_mss,speed_ms,0,blend_radius_m)
    |   movel([0.178198, -1.197569, -2.667162, -0.847658, 1.570796, 1.748994],accel_mss,speed_ms,0,blend_radius_m)
    |   movel([0.174052, -1.193011, -2.669332, -0.850046, 1.570796, 1.744849],accel_mss,speed_ms,0,blend_radius_m)
    |   speed_ms = 0.005
    |   movel([0.174052, -1.183660, -2.664472, -0.864257, 1.570796, 1.744849],accel_mss,speed_ms,0,blend_radius_m)
    |   speed_ms = 0.040
    |   movel([0.174973, -1.173939, -2.668970, -0.869480, 1.570796, 1.745769],accel_mss,speed_ms,0,blend_radius_m)
    |   speed_ms = 0.005
    |   movel([0.174973, -1.183317, -2.673872, -0.855200, 1.570796, 1.745769],accel_mss,speed_ms,0,blend_radius_m)
    |   speed_ms = 0.035
    |   movel([0.183391, -1.174965, -2.677704, -0.859720, 1.570796, 1.754187],accel_mss,speed_ms,0,blend_radius_m)
    |   movel([0.191503, -1.170447, -2.679746, -0.862196, 1.570796, 1.762299],accel_mss,speed_ms,0,blend_radius_m)
    |   # Splitting Linear movement in 2 (instruction 345: MoveL 242)
    |   movel([0.200392, -1.164034, -2.682608, -0.865747, 1.570796, 1.771188],accel_mss,speed_ms,0,blend_radius_m)
    |   movel([0.209367, -1.157593, -2.685440, -0.869356, 1.570796, 1.780164],accel_mss,speed_ms,0,blend_radius_m)
    |   speed_ms = 0.005
    |   # Splitting Linear movement in 6 (instruction 347: MoveL 243)
    |   movel([0.209367, -1.149712, -2.681263, -0.881414, 1.570796, 1.780164],accel_mss,speed_ms,0,blend_radius_m)
    |   movel([0.209367, -1.142010, -2.677050, -0.893329, 1.570796, 1.780164],accel_mss,speed_ms,0,blend_radius_m)
    |   movel([0.209367, -1.134485, -2.672802, -0.905102, 1.570796, 1.780164],accel_mss,speed_ms,0,blend_radius_m)
    |   movel([0.209367, -1.127133, -2.668520, -0.916736, 1.570796, 1.780164],accel_mss,speed_ms,0,blend_radius_m)
    |   movel([0.209367, -1.119952, -2.664204, -0.928233, 1.570796, 1.780164],accel_mss,speed_ms,0,blend_radius_m)
    |   movel([0.209367, -1.112939, -2.659855, -0.939595, 1.570796, 1.780164],accel_mss,speed_ms,0,blend_radius_m)
    |   speed_ms = 1.000
    |   movel([0.209367, -1.112939, -2.659855, -0.939595, 1.570796, 1.780164],accel_mss,speed_ms,0,blend_radius_m)
    |   # Splitting Linear movement in 20 (instruction 350: MoveL 245)
    |   movel([0.209367, -1.102727, -2.653272, -0.956390, 1.570796, 1.780164],accel_mss,speed_ms,0,blend_radius_m)
    |   movel([0.209367, -1.092877, -2.646619, -0.972893, 1.570796, 1.780164],accel_mss,speed_ms,0,blend_radius_m)
    |   movel([0.209367, -1.083379, -2.639898, -0.989111, 1.570796, 1.780164],accel_mss,speed_ms,0,blend_radius_m)
    |   movel([0.209367, -1.074224, -2.633112, -1.005052, 1.570796, 1.780164],accel_mss,speed_ms,0,blend_radius_m)
    |   movel([0.209367, -1.065403, -2.626263, -1.020723, 1.570796, 1.780164],accel_mss,speed_ms,0,blend_radius_m)
    |   movel([0.209367, -1.056906, -2.619352, -1.036130, 1.570796, 1.780164],accel_mss,speed_ms,0,blend_radius_m)
    |   movel([0.209367, -1.048725, -2.612382, -1.051281, 1.570796, 1.780164],accel_mss,speed_ms,0,blend_radius_m)
    |   movel([0.209367, -1.040851, -2.605355, -1.066183, 1.570796, 1.780164],accel_mss,speed_ms,0,blend_radius_m)
    |   movel([0.209367, -1.033275, -2.598271, -1.080843, 1.570796, 1.780164],accel_mss,speed_ms,0,blend_radius_m)
    |   movel([0.209367, -1.025989, -2.591132, -1.095267, 1.570796, 1.780164],accel_mss,speed_ms,0,blend_radius_m)
    |   movel([0.209367, -1.018985, -2.583941, -1.109462, 1.570796, 1.780164],accel_mss,speed_ms,0,blend_radius_m)
    |   movel([0.209367, -1.012256, -2.576699, -1.123435, 1.570796, 1.780164],accel_mss,speed_ms,0,blend_radius_m)
    |   movel([0.209367, -1.005792, -2.569406, -1.137191, 1.570796, 1.780164],accel_mss,speed_ms,0,blend_radius_m)
    |   movel([0.209367, -0.999587, -2.562064, -1.150738, 1.570796, 1.780164],accel_mss,speed_ms,0,blend_radius_m)
    |   movel([0.209367, -0.993633, -2.554675, -1.164081, 1.570796, 1.780164],accel_mss,speed_ms,0,blend_radius_m)
    |   movel([0.209367, -0.987924, -2.547240, -1.177225, 1.570796, 1.780164],accel_mss,speed_ms,0,blend_radius_m)
    |   movel([0.209367, -0.982452, -2.539759, -1.190178, 1.570796, 1.780164],accel_mss,speed_ms,0,blend_radius_m)
    |   movel([0.209367, -0.977210, -2.532234, -1.202944, 1.570796, 1.780164],accel_mss,speed_ms,0,blend_radius_m)
    |   movel([0.209367, -0.972193, -2.524666, -1.215530, 1.570796, 1.780164],accel_mss,speed_ms,0,blend_radius_m)
    |   movel([0.209367, -0.967394, -2.517056, -1.227940, 1.570796, 1.780164],accel_mss,speed_ms,0,blend_radius_m)
    |   # End of main program
    | end
    | 
    | Machining1()
